FUNCTION_BLOCK NewProductGUIFB (* JADE WORKER *)
  (* Standard: 61499-1 *)
  (* Version 1.0, 2014-04-22, Ahmed, Fraunhofer IGD *)
  (* Compiler header: package fb.rt; *)
  (* Compiler Java Sun JDK 1.5.0 *)
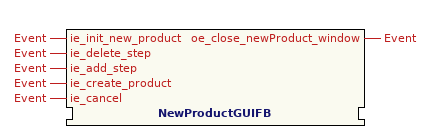
  EVENT_INPUT
    ie_init_new_product;
    ie_delete_step;
    ie_add_step;
    ie_create_product;
    ie_cancel;
  END_EVENT
  EVENT_OUTPUT
    oe_close_newProduct_window;
  END_EVENT
END_FUNCTION_BLOCK
